Fanuc KAREL source: kt00417.KL

-- PROVISIONAL review KL for V940-1; original PC SHA256 636fd7f9d877fb1d2ea436002f8cf8ec8dc0be971cfff5744f1d36ef5958b58c
-- Incomplete behavior may be omitted. Consult companion uncertainty JSON. Do not deploy.
PROGRAM KT00417
%NOLOCKGROUP
VAR
  OUT : BOOLEAN
-- UNRESOLVED_DECL H1 type=002017
-- UNRESOLVED_DECL Y2 type=002018
BEGIN
  -- V9_ZERO_TABLE_METADATA_HINT layout=0001; no indexed target words; source/name/runtime held
  -- UNRESOLVED_PC offsets 5-19; opcodes 2E,22,9D,33,B4
  -- UNRESOLVED_PC offsets 24-38; opcodes 2E,22,9D,33,B2
  -- UNRESOLVED_PC offsets 43-68; opcodes 22,9D,33,B3,22,9D,33,B1,5B,23
  -- UNRESOLVED_PC offsets 73-77; opcodes 7F
END KT00417
